TYPE ST_PositioningProfile :
STRUCT
	fPos : LREAL := 1.0; //[mm]
	fVel : LREAL := 1.0; //[mm/s]
	fAcc : LREAL := 1.0; //[mm/s^2]
	fDec : LREAL := 1.0; //[mm/s^2]
	fJrk : LREAL := 1.0; //[mm/s^3]
END_STRUCT
END_TYPE

(* stored: Version 1.1.0.1, ProductVersion 3.1.4024.12
   DUT ST_PositioningProfile: Id {83f008e9-e424-475b-ac6b-e0c4761275e2} *)
